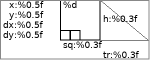
VISUALIZATION _VISU_MarkTriangle  // 150x60
VAR_IN_OUT
	mInst : ST_MarkDefinition;
END_VAR
    Rectangle (60,0 40x40), colour toggle: mInst.sState.bSet
        p874137650: mInst.fSqLength/mInst.fHeight*40-40
    Polygon (100,0) (100,40) (148,40), colour toggle: mInst.sState.bSet
        p3560616238: mInst.fSqLength/mInst.fHeight*40-40
    Rectangle (100,9 40x20), "h:%0.3f", tooltip "[m]", text variable: mInst.fHeight
        p3560616238: mInst.fSqLength/mInst.fHeight*40-40
    Rectangle (100,50 50x10), "tr:%0.3f", tooltip "[m]", text variable: mInst.fTrLength
        p3560616238: mInst.fSqLength/mInst.fHeight*40-40
    Rectangle (60,40 50x10), "sq:%0.3f", tooltip "[m]", text variable: mInst.fSqLength
    Rectangle (60,0 30x10), "%d", tooltip "Id", text variable: mInst.nId
    Rectangle (0,0 60x10), "x:%0.5f", tooltip "[m]", text variable: mInst.fPosX
    Rectangle (0,10 60x10), "y:%0.5f", tooltip "[m]", text variable: mInst.fPosY
    RoundedRectangle (60,30 10x10), tooltip "Missed", colour toggle: mInst.sState.bMissed, invisible if: NOT mInst.sState.bSet
    RoundedRectangle (70,30 10x10), tooltip "InArea", colour toggle: mInst.sState.bInArea, invisible if: NOT mInst.sState.bSet
    Rectangle (0,20 60x10), "dx:%0.5f", tooltip "[m]", text variable: mInst.sState.dx, invisible if: NOT mInst.sState.bSet
    Rectangle (0,30 60x10), "dy:%0.5f", tooltip "[m]", text variable: mInst.sState.dy, invisible if: NOT mInst.sState.bSet
END_VISUALIZATION

(* stored: Version 1.1.0.1, ProductVersion 3.1.4024.11
   Visu _VISU_MarkTriangle: Id {0965cb1c-3c98-4e76-8962-3f6f102112e7} *)
